// SIMATIC S7-200 SMART project (STEP 7-Micro/WIN SMART), CPU SR40

SYMBOL_TABLE USR1
下限位              I0.1
上限位              I0.2
右限位              I0.3
左限位              I0.4
上升按钮             I0.5
左行按钮             I0.6
松开按钮             I0.7
下降按钮             I1.0
右行按钮             I1.1
夹紧按钮             I1.2
手动开关             I2.0
回原点开关            I2.1
单步开关             I2.2
单周开关             I2.3
连续开关             I2.4
起动按钮             I2.6
停止按钮             I2.7
初始步              M0.0
原点条件             M0.5
转换允许             M0.6
连续标志             M0.7
A点降步             M2.0
夹紧步              M2.1
A点升步             M2.2
右行步              M2.3
B点降步             M2.4
松开步              M2.5
B点升步             M2.6
左行步              M2.7
下降阀              Q0.0
夹紧阀              Q0.1
上升阀              Q0.2
右行阀              Q0.3
左行阀              Q0.4
位置               VW2
END_SYMBOL_TABLE

ORGANIZATION_BLOCK MAIN:OB1
TITLE=PROGRAM COMMENTS
BEGIN
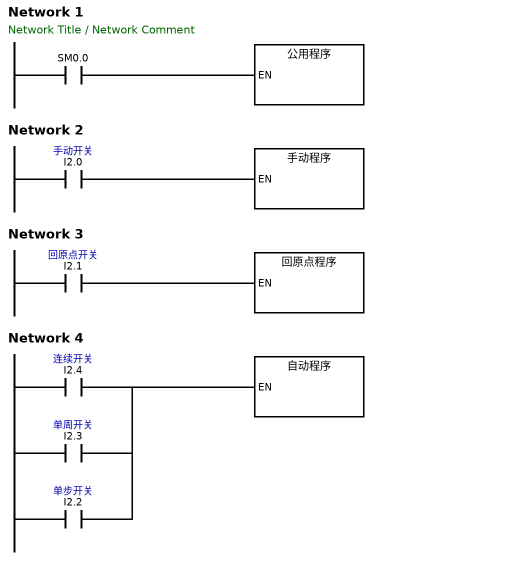
Network 1
// Network Title
// Network Comment
LD     SM0.0
CALL   公用程序:SBR0
Network 2
LD     手动开关:I2.0
CALL   手动程序:SBR1
Network 3
LD     回原点开关:I2.1
CALL   回原点程序:SBR2
Network 4
LD     连续开关:I2.4
O      单周开关:I2.3
O      单步开关:I2.2
CALL   自动程序:SBR3
END_ORGANIZATION_BLOCK

SUBROUTINE_BLOCK 公用程序:SBR0
TITLE=SUBROUTINE COMMENTS
BEGIN
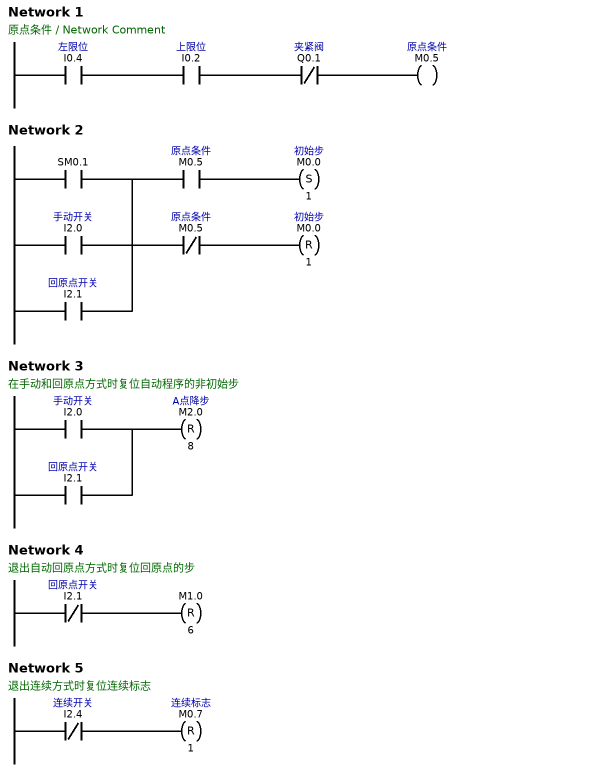
Network 1
// 原点条件
// Network Comment
LD     左限位:I0.4
A      上限位:I0.2
AN     夹紧阀:Q0.1
=      原点条件:M0.5
Network 2
LD     SM0.1
O      手动开关:I2.0
O      回原点开关:I2.1
LPS
A      原点条件:M0.5
S      初始步:M0.0, 1
LPP
AN     原点条件:M0.5
R      初始步:M0.0, 1
Network 3
// 在手动和回原点方式时复位自动程序的非初始步
LD     手动开关:I2.0
O      回原点开关:I2.1
R      A点降步:M2.0, 8
Network 4
// 退出自动回原点方式时复位回原点的步
LDN    回原点开关:I2.1
R      M1.0, 6
Network 5
// 退出连续方式时复位连续标志
LDN    连续开关:I2.4
R      连续标志:M0.7, 1
END_SUBROUTINE_BLOCK

SUBROUTINE_BLOCK 手动程序:SBR1
TITLE=SUBROUTINE COMMENTS
BEGIN
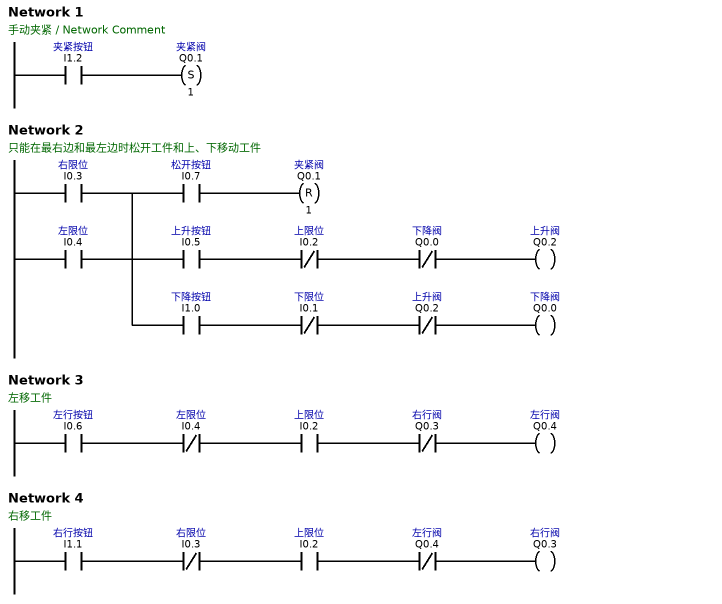
Network 1
// 手动夹紧
// Network Comment
LD     夹紧按钮:I1.2
S      夹紧阀:Q0.1, 1
Network 2
// 只能在最右边和最左边时松开工件和上、下移动工件
LD     右限位:I0.3
O      左限位:I0.4
LPS
A      松开按钮:I0.7
R      夹紧阀:Q0.1, 1
LRD
A      上升按钮:I0.5
AN     上限位:I0.2
AN     下降阀:Q0.0
=      上升阀:Q0.2
LPP
A      下降按钮:I1.0
AN     下限位:I0.1
AN     上升阀:Q0.2
=      下降阀:Q0.0
Network 3
// 左移工件
LD     左行按钮:I0.6
AN     左限位:I0.4
A      上限位:I0.2
AN     右行阀:Q0.3
=      左行阀:Q0.4
Network 4
// 右移工件
LD     右行按钮:I1.1
AN     右限位:I0.3
A      上限位:I0.2
AN     左行阀:Q0.4
=      右行阀:Q0.3
Network 5
// Network Title
// Network Comment
END_SUBROUTINE_BLOCK

SUBROUTINE_BLOCK 回原点程序:SBR2
TITLE=SUBROUTINE COMMENTS
BEGIN
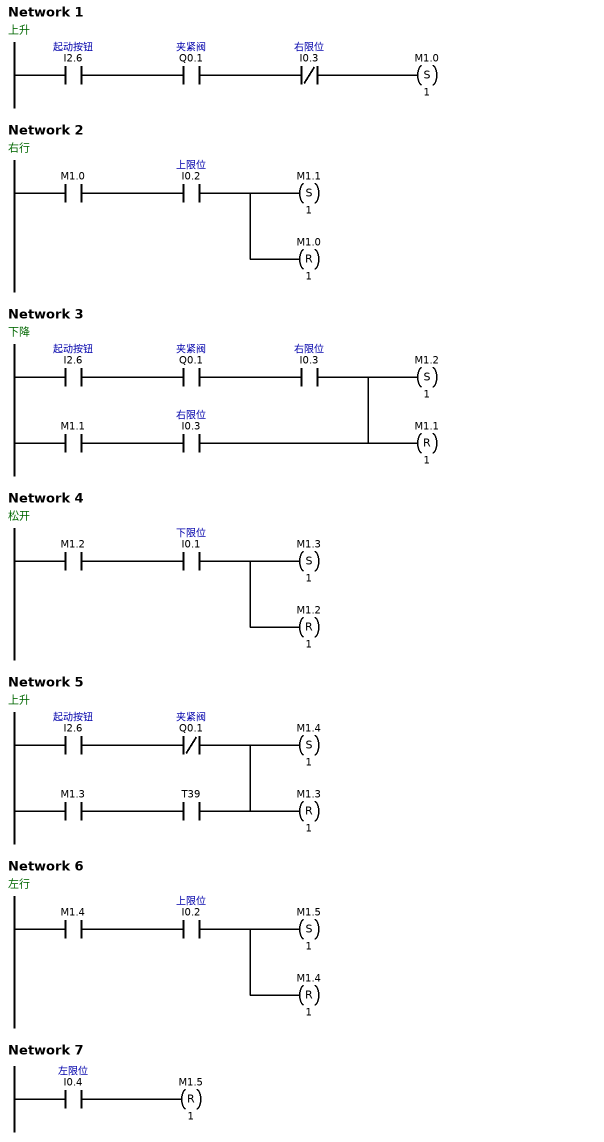
Network 1
// 上升
LD     起动按钮:I2.6
A      夹紧阀:Q0.1
AN     右限位:I0.3
S      M1.0, 1
Network 2
// 右行
LD     M1.0
A      上限位:I0.2
S      M1.1, 1
R      M1.0, 1
Network 3
// 下降
LD     起动按钮:I2.6
A      夹紧阀:Q0.1
A      右限位:I0.3
LD     M1.1
A      右限位:I0.3
OLD
S      M1.2, 1
R      M1.1, 1
Network 4
// 松开
LD     M1.2
A      下限位:I0.1
S      M1.3, 1
R      M1.2, 1
Network 5
// 上升
LD     起动按钮:I2.6
AN     夹紧阀:Q0.1
LD     M1.3
A      T39
OLD
S      M1.4, 1
R      M1.3, 1
Network 6
// 左行
LD     M1.4
A      上限位:I0.2
S      M1.5, 1
R      M1.4, 1
Network 7
LD     左限位:I0.4
R      M1.5, 1
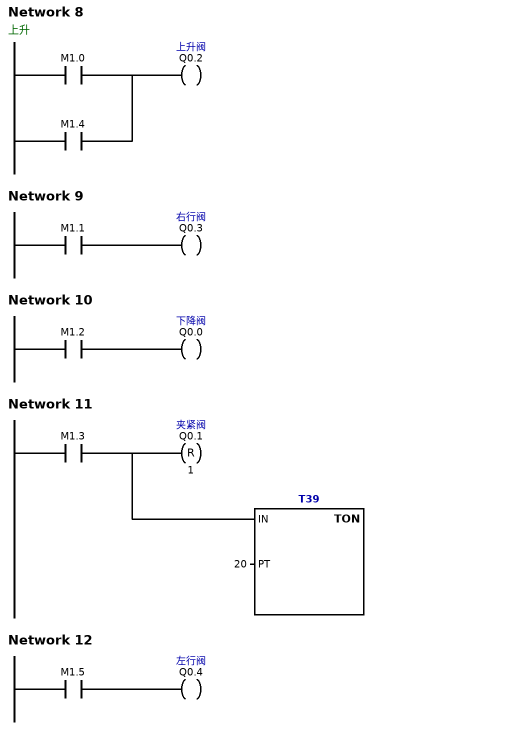
Network 8
// 上升
LD     M1.0
O      M1.4
=      上升阀:Q0.2
Network 9
LD     M1.1
=      右行阀:Q0.3
Network 10
LD     M1.2
=      下降阀:Q0.0
Network 11
LD     M1.3
R      夹紧阀:Q0.1, 1
TON    T39, 20
Network 12
LD     M1.5
=      左行阀:Q0.4
END_SUBROUTINE_BLOCK

SUBROUTINE_BLOCK 自动程序:SBR3
TITLE=SUBROUTINE COMMENTS
BEGIN
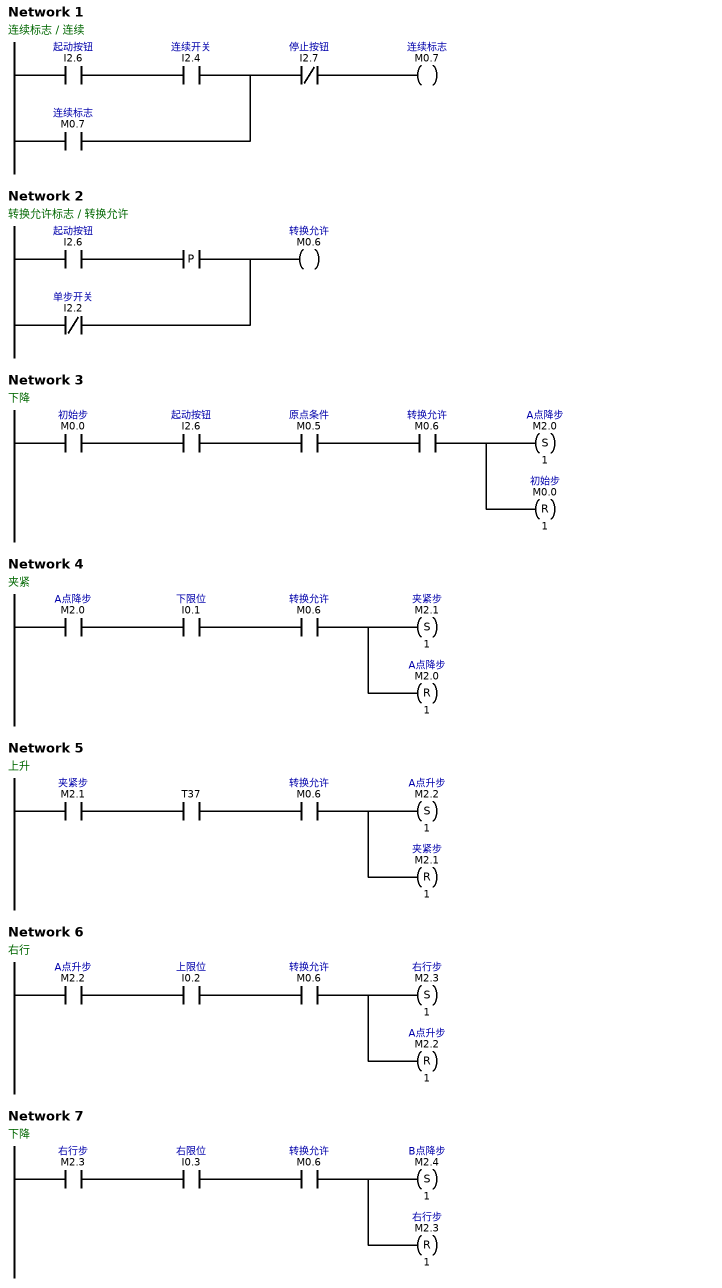
Network 1
// 连续标志
// 连续
LD     起动按钮:I2.6
A      连续开关:I2.4
O      连续标志:M0.7
AN     停止按钮:I2.7
=      连续标志:M0.7
Network 2
// 转换允许标志
// 转换允许
LD     起动按钮:I2.6
EU
ON     单步开关:I2.2
=      转换允许:M0.6
Network 3
// 下降
LD     初始步:M0.0
A      起动按钮:I2.6
A      原点条件:M0.5
A      转换允许:M0.6
S      A点降步:M2.0, 1
R      初始步:M0.0, 1
Network 4
// 夹紧
LD     A点降步:M2.0
A      下限位:I0.1
A      转换允许:M0.6
S      夹紧步:M2.1, 1
R      A点降步:M2.0, 1
Network 5
// 上升
LD     夹紧步:M2.1
A      T37
A      转换允许:M0.6
S      A点升步:M2.2, 1
R      夹紧步:M2.1, 1
Network 6
// 右行
LD     A点升步:M2.2
A      上限位:I0.2
A      转换允许:M0.6
S      右行步:M2.3, 1
R      A点升步:M2.2, 1
Network 7
// 下降
LD     右行步:M2.3
A      右限位:I0.3
A      转换允许:M0.6
S      B点降步:M2.4, 1
R      右行步:M2.3, 1
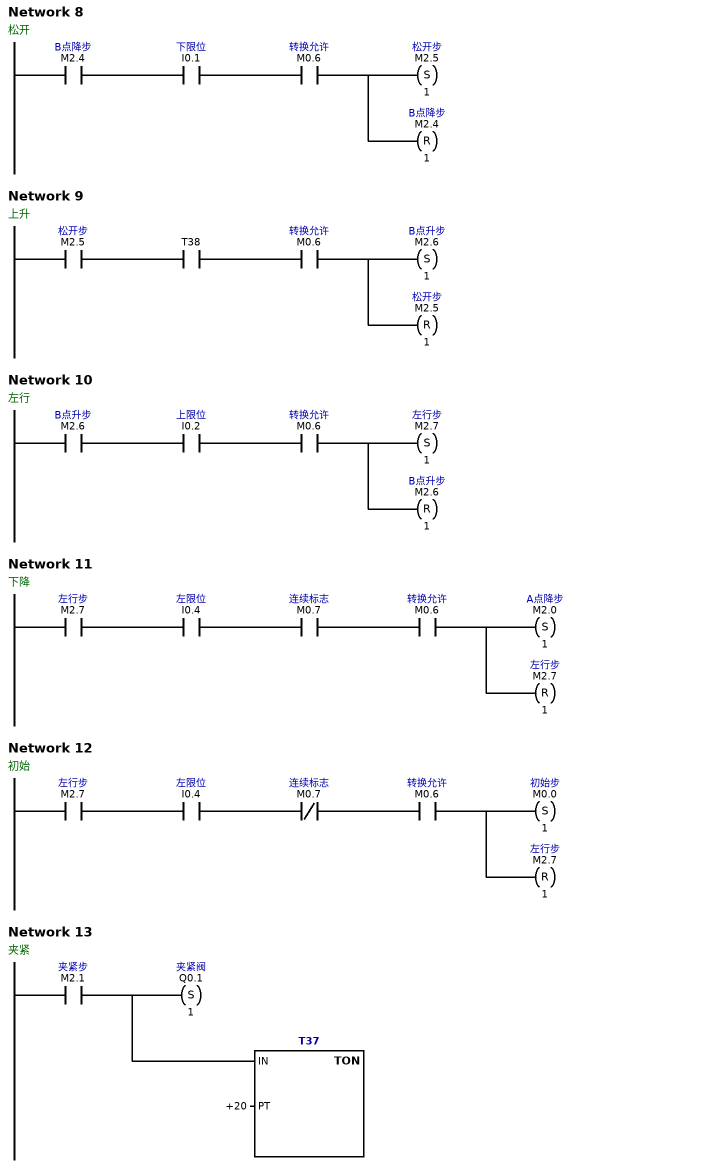
Network 8
// 松开
LD     B点降步:M2.4
A      下限位:I0.1
A      转换允许:M0.6
S      松开步:M2.5, 1
R      B点降步:M2.4, 1
Network 9
// 上升
LD     松开步:M2.5
A      T38
A      转换允许:M0.6
S      B点升步:M2.6, 1
R      松开步:M2.5, 1
Network 10
// 左行
LD     B点升步:M2.6
A      上限位:I0.2
A      转换允许:M0.6
S      左行步:M2.7, 1
R      B点升步:M2.6, 1
Network 11
// 下降
LD     左行步:M2.7
A      左限位:I0.4
A      连续标志:M0.7
A      转换允许:M0.6
S      A点降步:M2.0, 1
R      左行步:M2.7, 1
Network 12
// 初始
LD     左行步:M2.7
A      左限位:I0.4
AN     连续标志:M0.7
A      转换允许:M0.6
S      初始步:M0.0, 1
R      左行步:M2.7, 1
Network 13
// 夹紧
LD     夹紧步:M2.1
S      夹紧阀:Q0.1, 1
TON    T37, +20
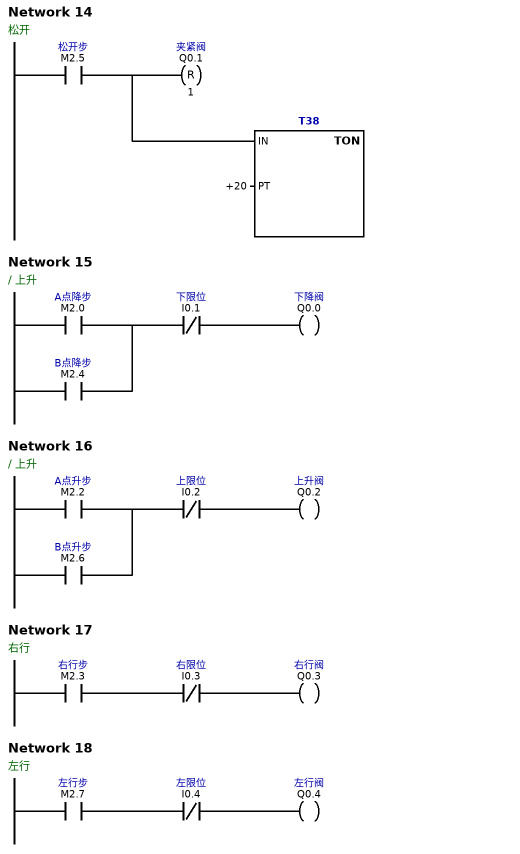
Network 14
// 松开
LD     松开步:M2.5
R      夹紧阀:Q0.1, 1
TON    T38, +20
Network 15
//  
// 上升
LD     A点降步:M2.0
O      B点降步:M2.4
AN     下限位:I0.1
=      下降阀:Q0.0
Network 16
//  
// 上升
LD     A点升步:M2.2
O      B点升步:M2.6
AN     上限位:I0.2
=      上升阀:Q0.2
Network 17
// 右行
LD     右行步:M2.3
AN     右限位:I0.3
=      右行阀:Q0.3
Network 18
// 左行
LD     左行步:M2.7
AN     左限位:I0.4
=      左行阀:Q0.4
END_SUBROUTINE_BLOCK

DATA_BLOCK_TAB 用户定义1
BEGIN
//DATA BLOCK COMMENTS
//Press F1 for help and example data block
         位置, 1000
END_DATA_BLOCK_TAB
